Omron CX-Programmer project NewProject (CX-Programmer 9.80)

# PLC NewPLC1: CQM1 CPU41

## Program NewProgram1 (no task)

### Section Section1

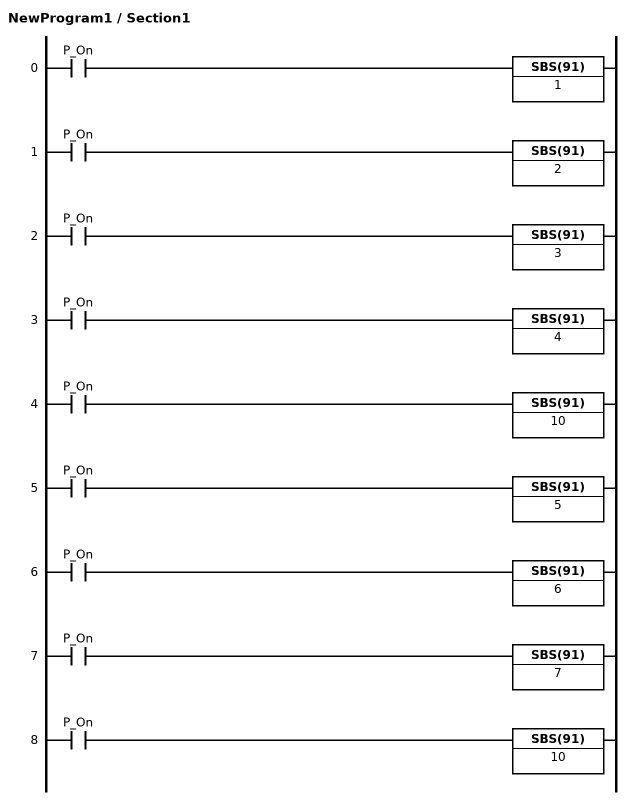
; rung 0
LD P_On
SBS(91) 1
; rung 1
LD P_On
SBS(91) 2
; rung 2
LD P_On
SBS(91) 3
; rung 3
LD P_On
SBS(91) 4
; rung 4
LD P_On
SBS(91) 10
; rung 5
LD P_On
SBS(91) 5
; rung 6
LD P_On
SBS(91) 6
; rung 7
LD P_On
SBS(91) 7
; rung 8
LD P_On
SBS(91) 10

### Section Section2

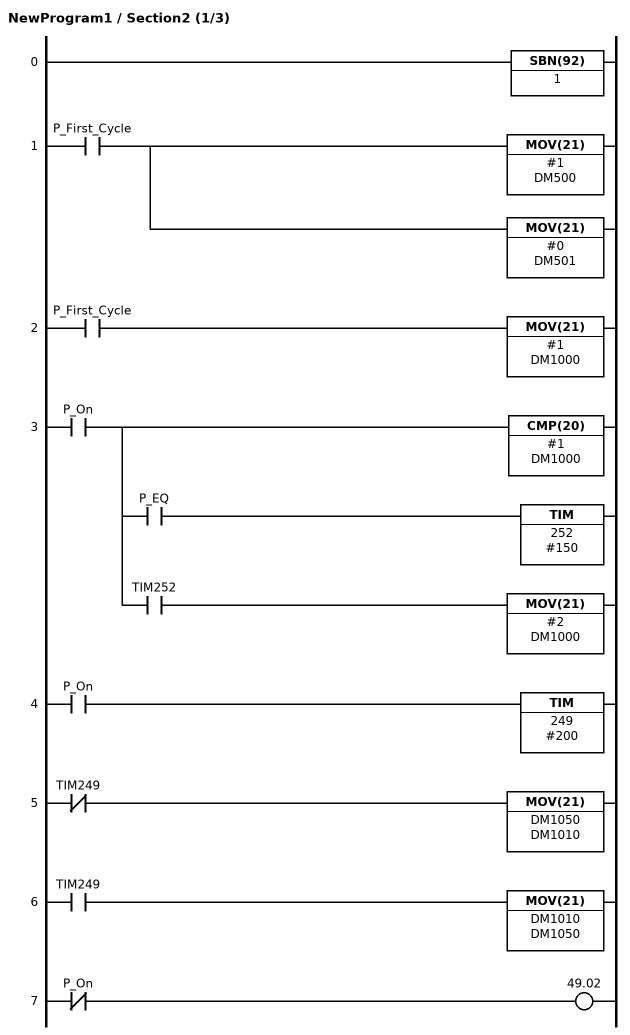
; rung 0
SBN(92) 1
; rung 1
LD P_First_Cycle
MOV(21) #1 DM500
MOV(21) #0 DM501
; rung 2
LD P_First_Cycle
MOV(21) #1 DM1000
; rung 3
LD P_On
OUT TR0
CMP(20) #1 DM1000
AND P_EQ
TIM 252 #150
LD TR0
AND TIM252
MOV(21) #2 DM1000
; rung 4
LD P_On
TIM 249 #200
; rung 5
LDNOT TIM249
MOV(21) DM1050 DM1010
; rung 6
LD TIM249
MOV(21) DM1010 DM1050
; rung 7
LDNOT P_On
OUT 49.02

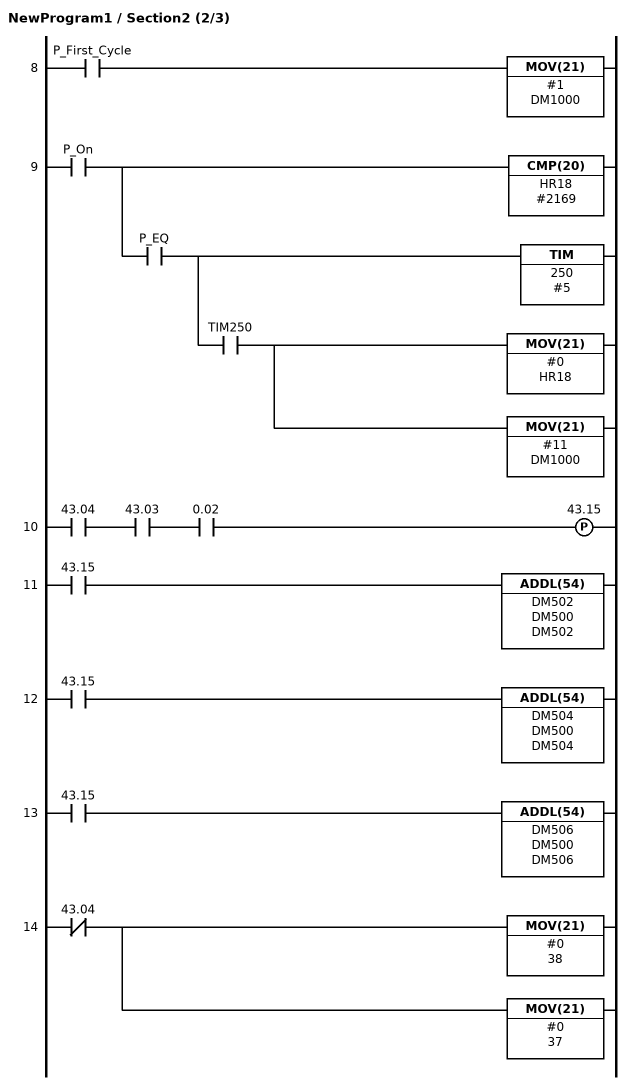
; rung 8
LD P_First_Cycle
MOV(21) #1 DM1000
; rung 9
LD P_On
CMP(20) HR18 #2169
AND P_EQ
TIM 250 #5
AND TIM250
MOV(21) #0 HR18
MOV(21) #11 DM1000
; rung 10
LD 43.04
AND 43.03
AND 0.02
DIFU(13) 43.15
; rung 11
LD 43.15
ADDL(54) DM502 DM500 DM502
; rung 12
LD 43.15
ADDL(54) DM504 DM500 DM504
; rung 13
LD 43.15
ADDL(54) DM506 DM500 DM506
; rung 14
LDNOT 43.04
MOV(21) #0 38
MOV(21) #0 37

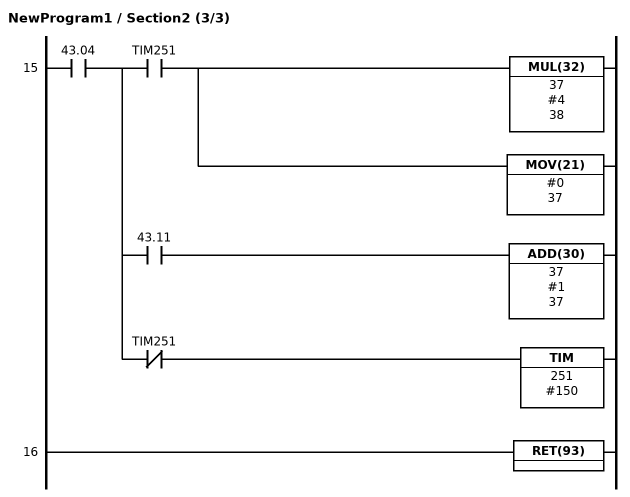
; rung 15
LD 43.04
OUT TR0
AND TIM251
MUL(32) 37 #4 38
MOV(21) #0 37
LD TR0
AND 43.11
ADD(30) 37 #1 37
LD TR0
ANDNOT TIM251
TIM 251 #150
; rung 16
RET(93)

### Section Section3

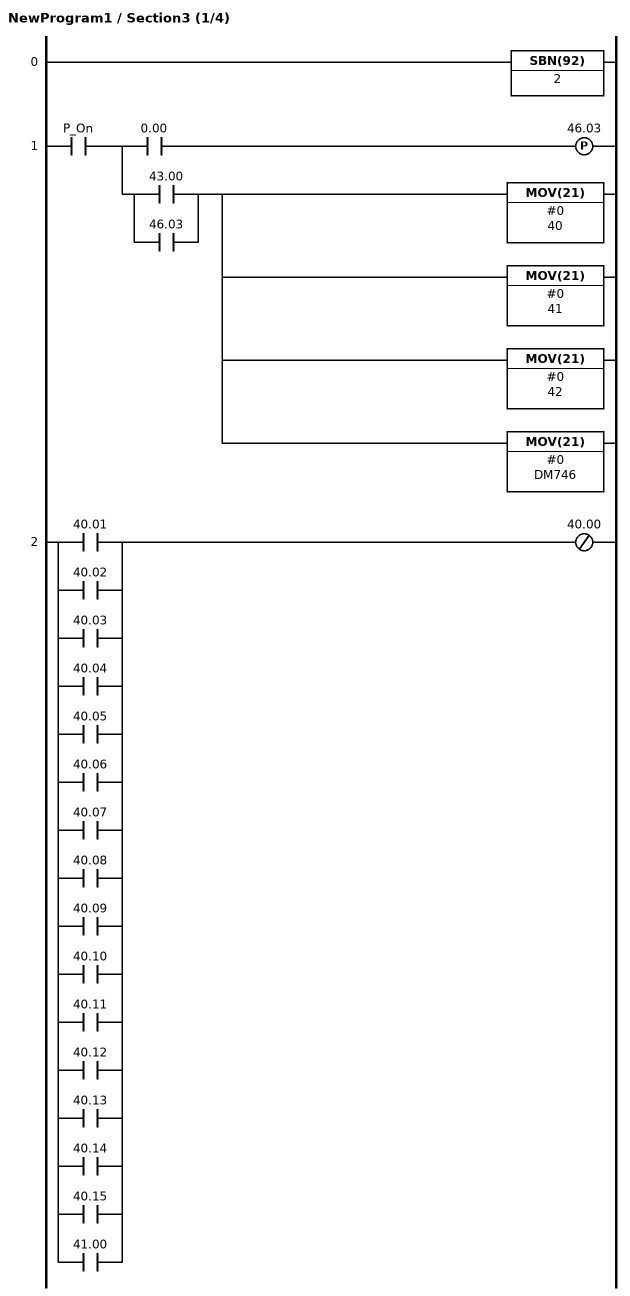
; rung 0
SBN(92) 2
; rung 1
LD P_On
OUT TR0
AND 0.00
DIFU(13) 46.03
LD TR0
LD 43.00
OR 46.03
ANDLD
MOV(21) #0 40
MOV(21) #0 41
MOV(21) #0 42
MOV(21) #0 DM746
; rung 2
LD 40.01
OR 40.02
OR 40.03
OR 40.04
OR 40.05
OR 40.06
OR 40.07
OR 40.08
OR 40.09
OR 40.10
OR 40.11
OR 40.12
OR 40.13
OR 40.14
OR 40.15
OR 41.00
OUTNOT 40.00

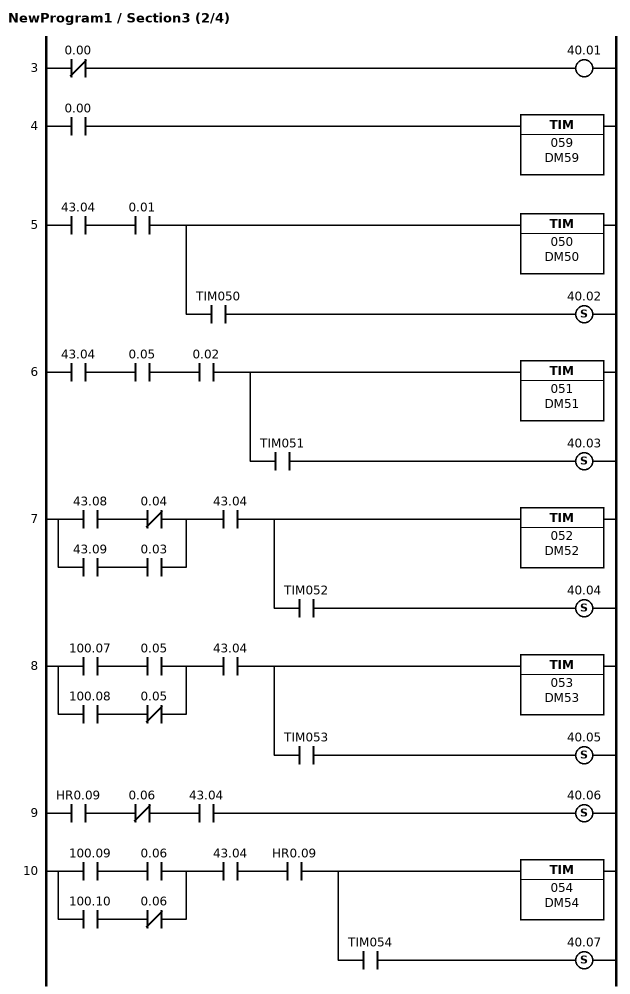
; rung 3
LDNOT 0.00
OUT 40.01
; rung 4
LD 0.00
TIM 059 DM59
; rung 5
LD 43.04
AND 0.01
TIM 050 DM50
AND TIM050
SET 40.02
; rung 6
LD 43.04
AND 0.05
AND 0.02
TIM 051 DM51
AND TIM051
SET 40.03
; rung 7
LD 43.08
ANDNOT 0.04
LD 43.09
AND 0.03
ORLD
AND 43.04
TIM 052 DM52
AND TIM052
SET 40.04
; rung 8
LD 100.07
AND 0.05
LD 100.08
ANDNOT 0.05
ORLD
AND 43.04
TIM 053 DM53
AND TIM053
SET 40.05
; rung 9
LD HR0.09
ANDNOT 0.06
AND 43.04
SET 40.06
; rung 10
LD 100.09
AND 0.06
LD 100.10
ANDNOT 0.06
ORLD
AND 43.04
AND HR0.09
TIM 054 DM54
AND TIM054
SET 40.07

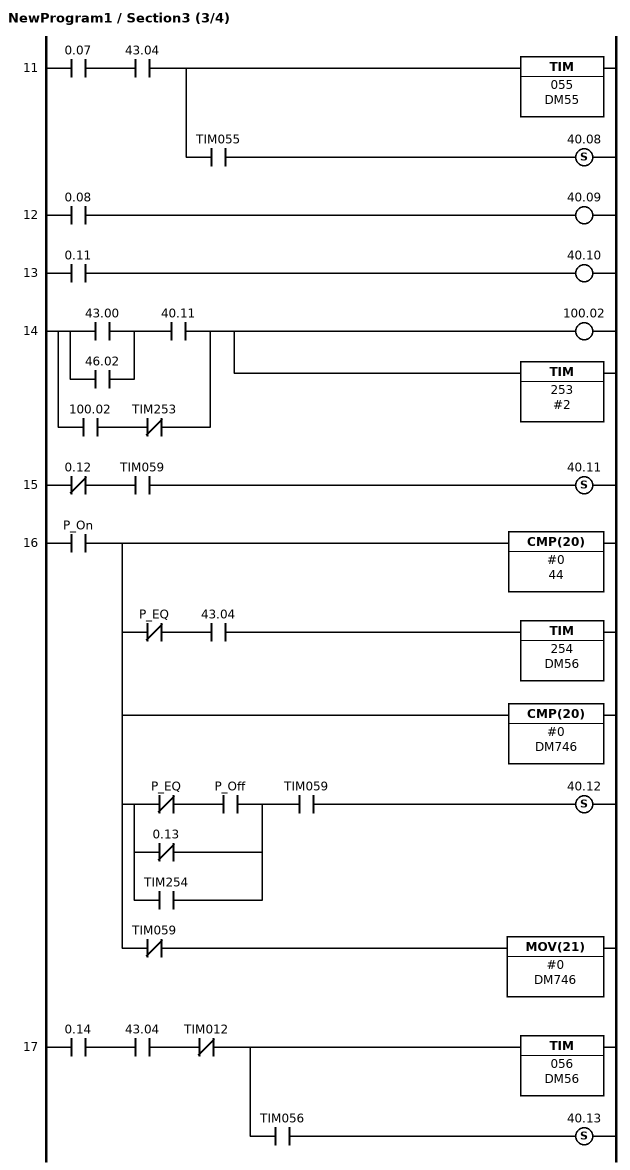
; rung 11
LD 0.07
AND 43.04
TIM 055 DM55
AND TIM055
SET 40.08
; rung 12
LD 0.08
OUT 40.09
; rung 13
LD 0.11
OUT 40.10
; rung 14
LD 43.00
OR 46.02
AND 40.11
LD 100.02
ANDNOT TIM253
ORLD
OUT 100.02
TIM 253 #2
; rung 15
LDNOT 0.12
AND TIM059
SET 40.11
; rung 16
LD P_On
OUT TR0
CMP(20) #0 44
ANDNOT P_EQ
AND 43.04
TIM 254 DM56
LD TR0
CMP(20) #0 DM746
LDNOT P_EQ
AND P_Off
ORNOT 0.13
OR TIM254
ANDLD
AND TIM059
SET 40.12
LD TR0
ANDNOT TIM059
MOV(21) #0 DM746
; rung 17
LD 0.14
AND 43.04
ANDNOT TIM012
TIM 056 DM56
AND TIM056
SET 40.13

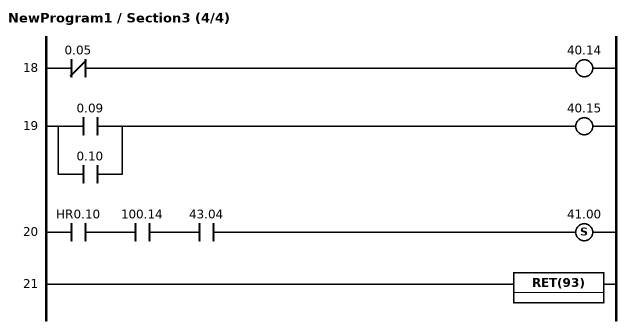
; rung 18
LDNOT 0.05
OUT 40.14
; rung 19
LD 0.09
OR 0.10
OUT 40.15
; rung 20
LD HR0.10
AND 100.14
AND 43.04
SET 41.00
; rung 21
RET(93)

### Section Section4

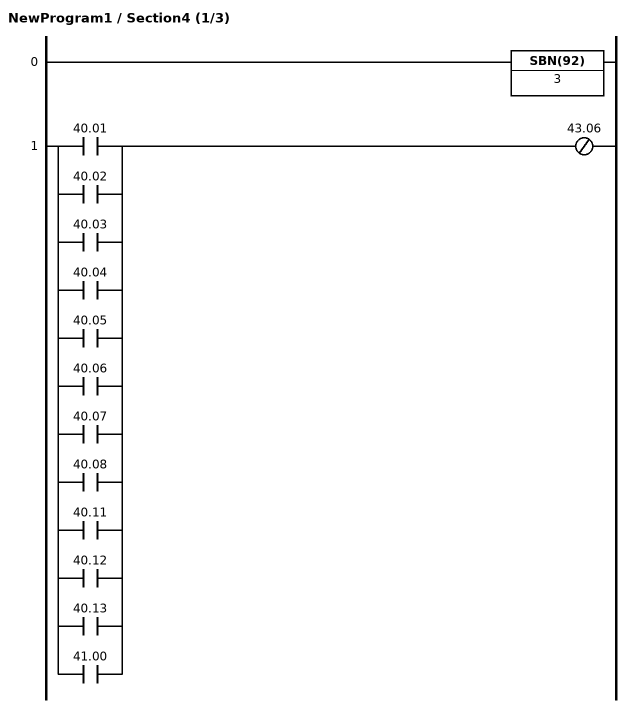
; rung 0
SBN(92) 3
; rung 1
LD 40.01
OR 40.02
OR 40.03
OR 40.04
OR 40.05
OR 40.06
OR 40.07
OR 40.08
OR 40.11
OR 40.12
OR 40.13
OR 41.00
OUTNOT 43.06

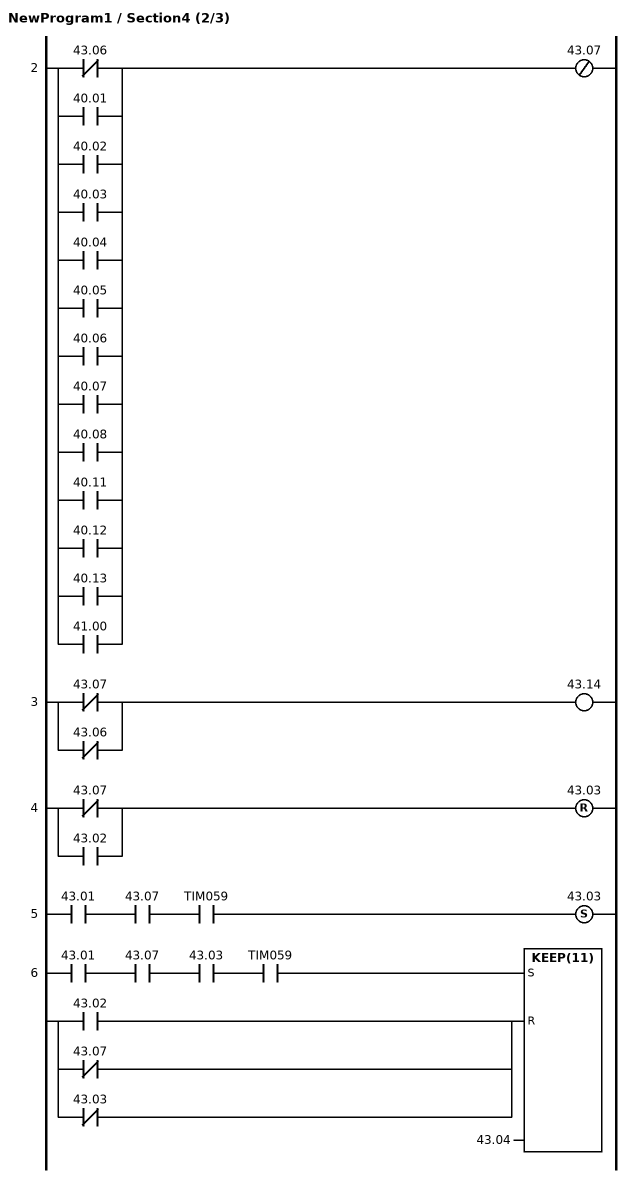
; rung 2
LDNOT 43.06
OR 40.01
OR 40.02
OR 40.03
OR 40.04
OR 40.05
OR 40.06
OR 40.07
OR 40.08
OR 40.11
OR 40.12
OR 40.13
OR 41.00
OUTNOT 43.07
; rung 3
LDNOT 43.07
ORNOT 43.06
OUT 43.14
; rung 4
LDNOT 43.07
OR 43.02
RSET 43.03
; rung 5
LD 43.01
AND 43.07
AND TIM059
SET 43.03
; rung 6
LD 43.01
AND 43.07
AND 43.03
AND TIM059
LD 43.02
ORNOT 43.07
ORNOT 43.03
KEEP(11) 43.04

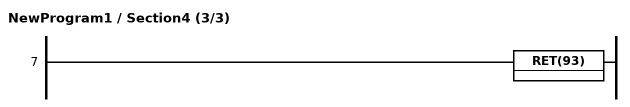
; rung 7
RET(93)

### Section Section5

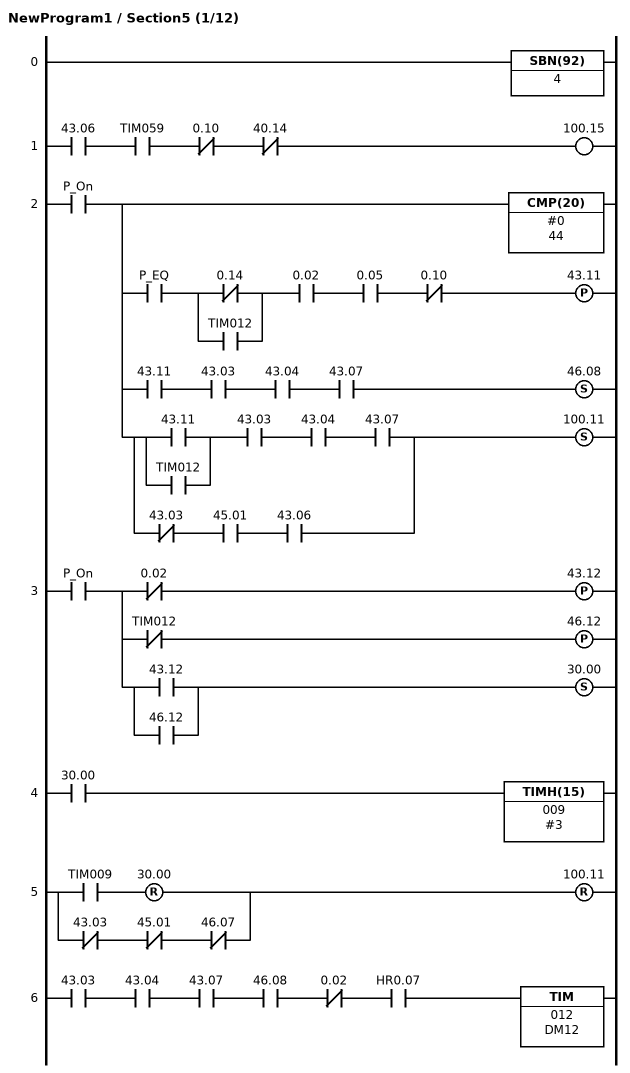
; rung 0
SBN(92) 4
; rung 1
LD 43.06
AND TIM059
ANDNOT 0.10
ANDNOT 40.14
OUT 100.15
; rung 2
LD P_On
OUT TR0
CMP(20) #0 44
AND P_EQ
LDNOT 0.14
OR TIM012
ANDLD
AND 0.02
AND 0.05
ANDNOT 0.10
DIFU(13) 43.11
LD TR0
AND 43.11
AND 43.03
AND 43.04
AND 43.07
SET 46.08
LD TR0
LD 43.11
OR TIM012
AND 43.03
AND 43.04
AND 43.07
LDNOT 43.03
AND 45.01
AND 43.06
ORLD
ANDLD
SET 100.11
; rung 3
LD P_On
OUT TR0
ANDNOT 0.02
DIFU(13) 43.12
LD TR0
ANDNOT TIM012
DIFU(13) 46.12
LD TR0
LD 43.12
OR 46.12
ANDLD
SET 30.00
; rung 4
LD 30.00
TIMH(15) 009 #3
; rung 5
LD TIM009
RSET 30.00
LDNOT 43.03
ANDNOT 45.01
ANDNOT 46.07
ORLD
RSET 100.11
; rung 6
LD 43.03
AND 43.04
AND 43.07
AND 46.08
ANDNOT 0.02
AND HR0.07
TIM 012 DM12

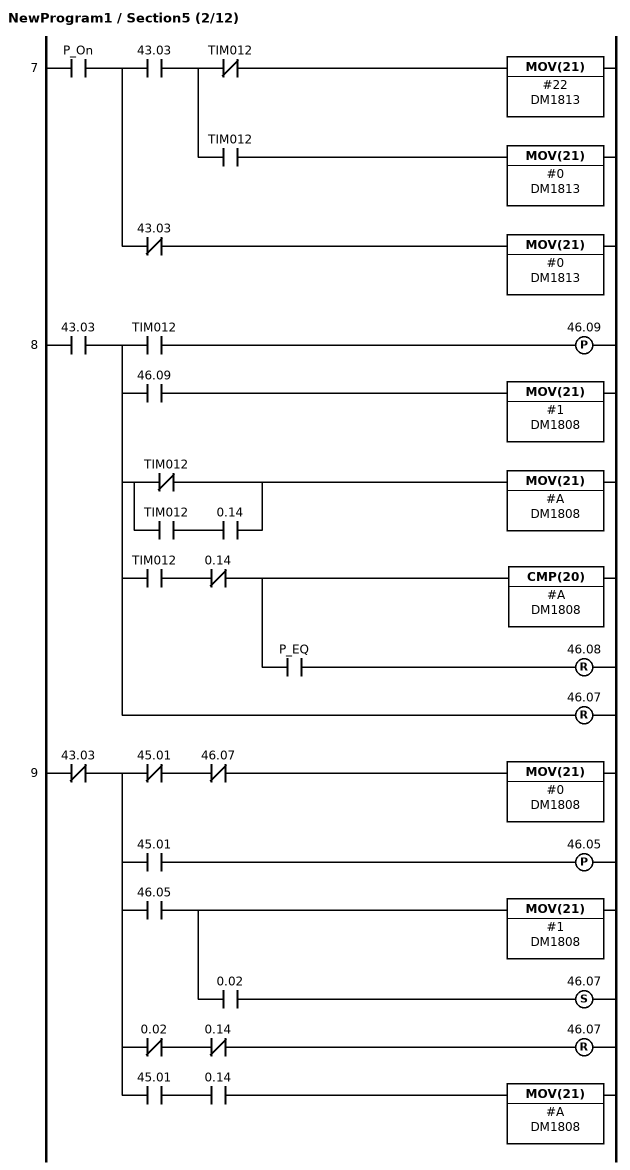
; rung 7
LD P_On
OUT TR0
AND 43.03
OUT TR1
ANDNOT TIM012
MOV(21) #22 DM1813
LD TR1
AND TIM012
MOV(21) #0 DM1813
LD TR0
ANDNOT 43.03
MOV(21) #0 DM1813
; rung 8
LD 43.03
OUT TR0
AND TIM012
DIFU(13) 46.09
LD TR0
AND 46.09
MOV(21) #1 DM1808
LD TR0
LDNOT TIM012
LD TIM012
AND 0.14
ORLD
ANDLD
MOV(21) #A DM1808
LD TR0
AND TIM012
ANDNOT 0.14
CMP(20) #A DM1808
AND P_EQ
RSET 46.08
LD TR0
RSET 46.07
; rung 9
LDNOT 43.03
OUT TR0
ANDNOT 45.01
ANDNOT 46.07
MOV(21) #0 DM1808
LD TR0
AND 45.01
DIFU(13) 46.05
LD TR0
AND 46.05
MOV(21) #1 DM1808
AND 0.02
SET 46.07
LD TR0
ANDNOT 0.02
ANDNOT 0.14
RSET 46.07
LD TR0
AND 45.01
AND 0.14
MOV(21) #A DM1808

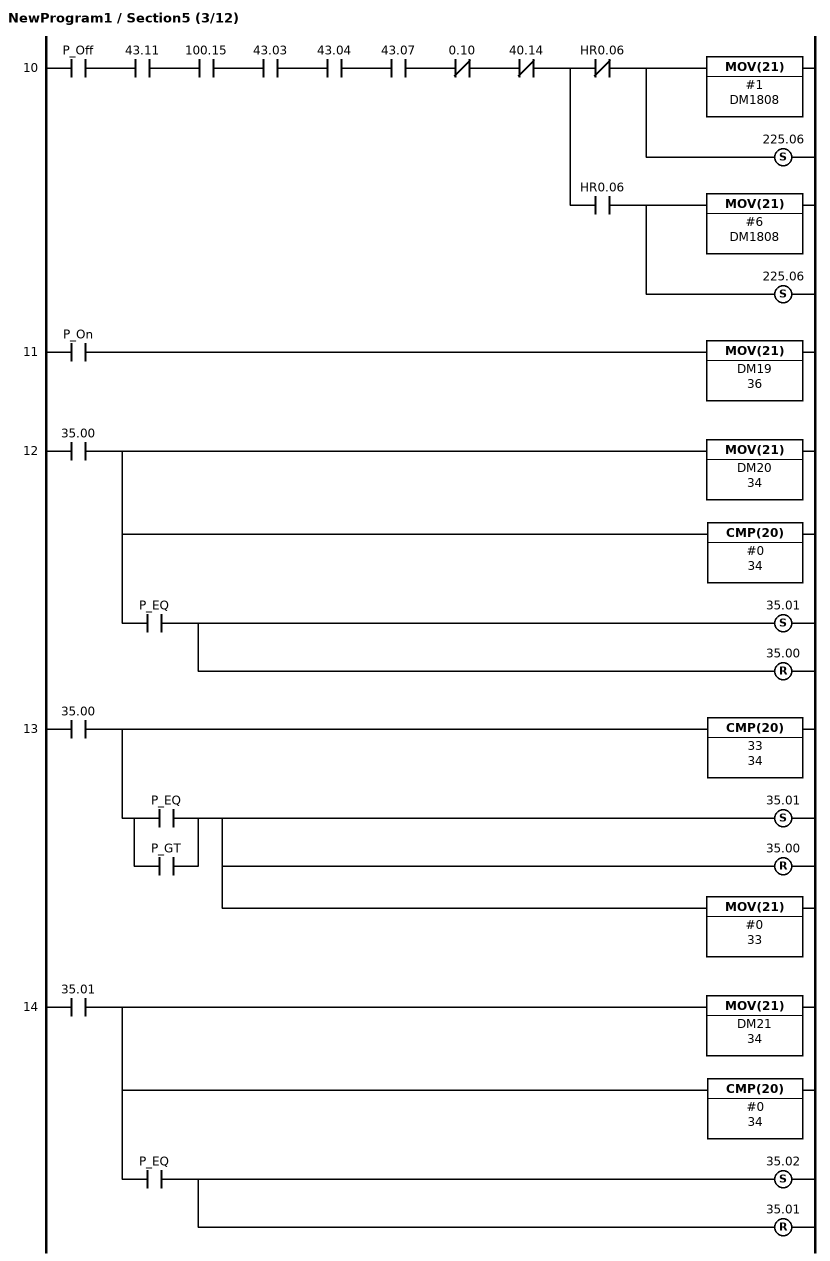
; rung 10
LD P_Off
AND 43.11
AND 100.15
AND 43.03
AND 43.04
AND 43.07
ANDNOT 0.10
ANDNOT 40.14
OUT TR0
ANDNOT HR0.06
MOV(21) #1 DM1808
SET 225.06
LD TR0
AND HR0.06
MOV(21) #6 DM1808
SET 225.06
; rung 11
LD P_On
MOV(21) DM19 36
; rung 12
LD 35.00
MOV(21) DM20 34
CMP(20) #0 34
AND P_EQ
SET 35.01
RSET 35.00
; rung 13
LD 35.00
CMP(20) 33 34
LD P_EQ
OR P_GT
ANDLD
SET 35.01
RSET 35.00
MOV(21) #0 33
; rung 14
LD 35.01
MOV(21) DM21 34
CMP(20) #0 34
AND P_EQ
SET 35.02
RSET 35.01

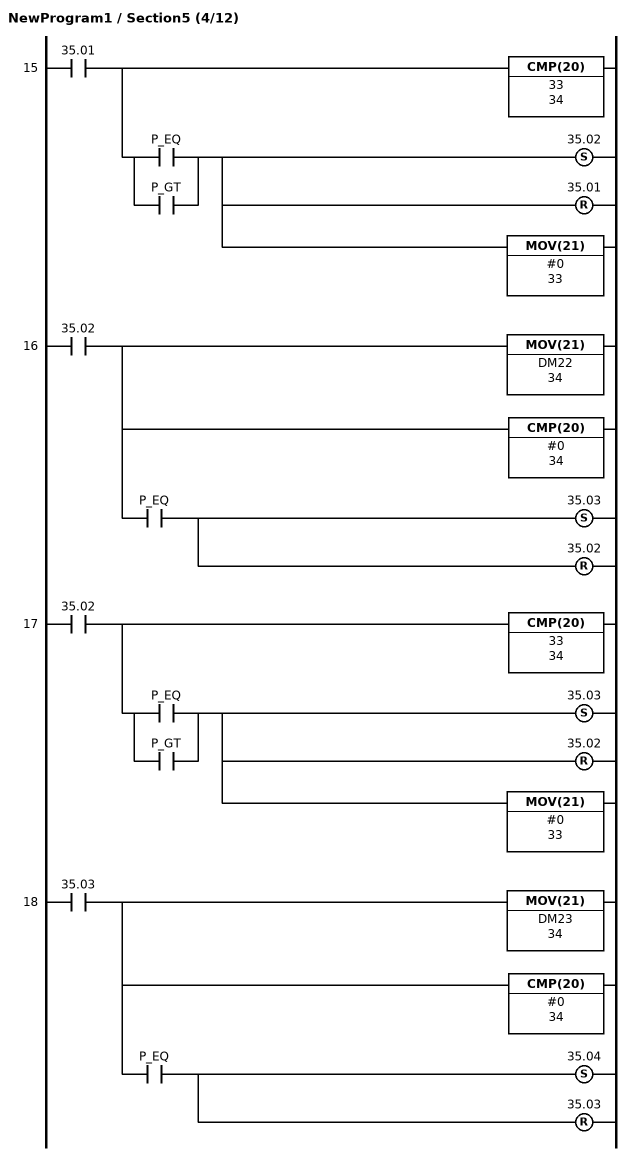
; rung 15
LD 35.01
CMP(20) 33 34
LD P_EQ
OR P_GT
ANDLD
SET 35.02
RSET 35.01
MOV(21) #0 33
; rung 16
LD 35.02
MOV(21) DM22 34
CMP(20) #0 34
AND P_EQ
SET 35.03
RSET 35.02
; rung 17
LD 35.02
CMP(20) 33 34
LD P_EQ
OR P_GT
ANDLD
SET 35.03
RSET 35.02
MOV(21) #0 33
; rung 18
LD 35.03
MOV(21) DM23 34
CMP(20) #0 34
AND P_EQ
SET 35.04
RSET 35.03

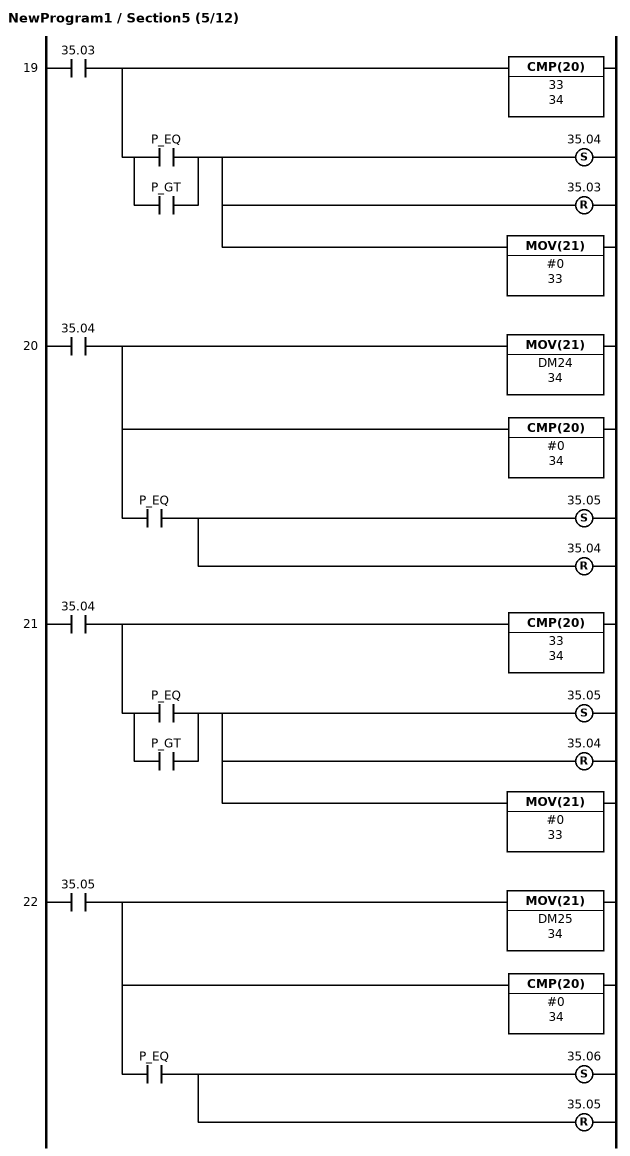
; rung 19
LD 35.03
CMP(20) 33 34
LD P_EQ
OR P_GT
ANDLD
SET 35.04
RSET 35.03
MOV(21) #0 33
; rung 20
LD 35.04
MOV(21) DM24 34
CMP(20) #0 34
AND P_EQ
SET 35.05
RSET 35.04
; rung 21
LD 35.04
CMP(20) 33 34
LD P_EQ
OR P_GT
ANDLD
SET 35.05
RSET 35.04
MOV(21) #0 33
; rung 22
LD 35.05
MOV(21) DM25 34
CMP(20) #0 34
AND P_EQ
SET 35.06
RSET 35.05

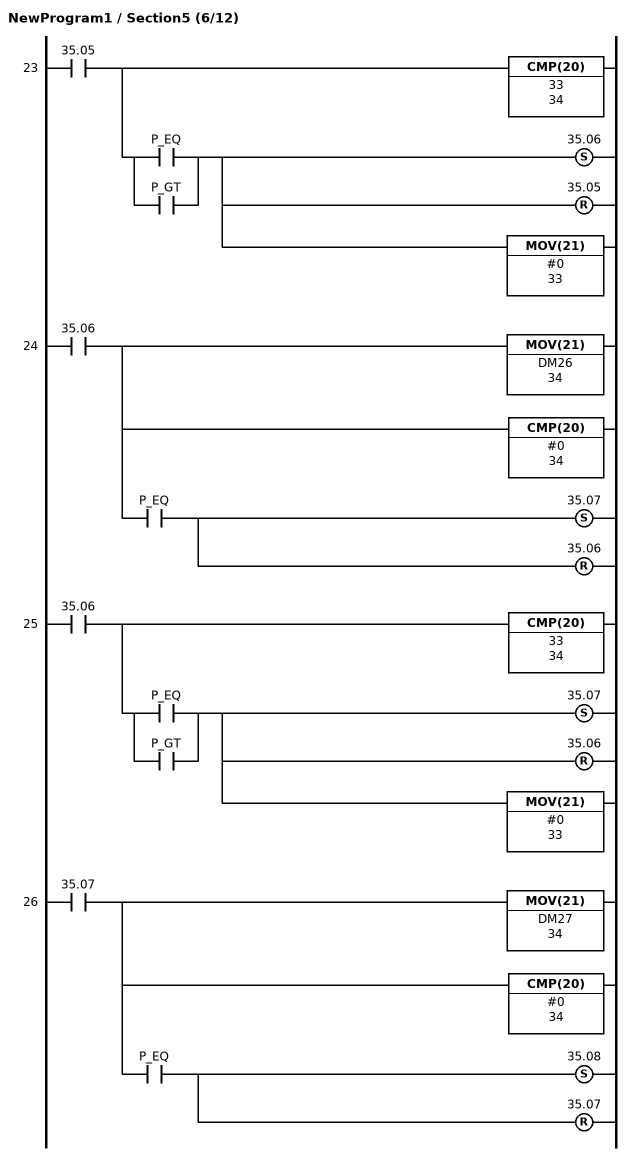
; rung 23
LD 35.05
CMP(20) 33 34
LD P_EQ
OR P_GT
ANDLD
SET 35.06
RSET 35.05
MOV(21) #0 33
; rung 24
LD 35.06
MOV(21) DM26 34
CMP(20) #0 34
AND P_EQ
SET 35.07
RSET 35.06
; rung 25
LD 35.06
CMP(20) 33 34
LD P_EQ
OR P_GT
ANDLD
SET 35.07
RSET 35.06
MOV(21) #0 33
; rung 26
LD 35.07
MOV(21) DM27 34
CMP(20) #0 34
AND P_EQ
SET 35.08
RSET 35.07

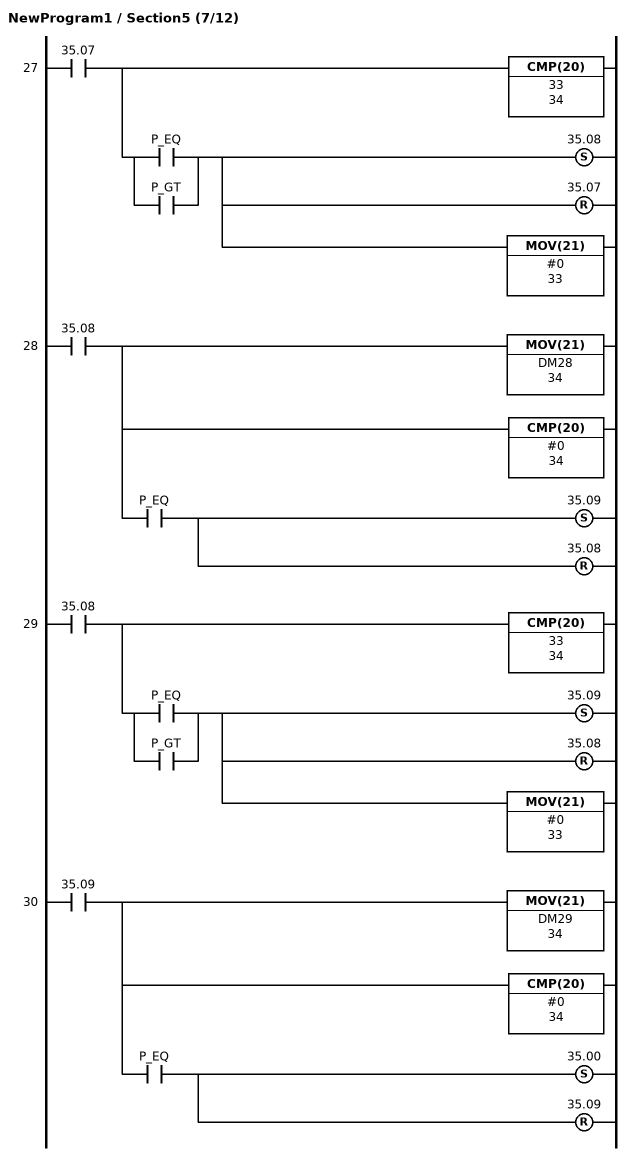
; rung 27
LD 35.07
CMP(20) 33 34
LD P_EQ
OR P_GT
ANDLD
SET 35.08
RSET 35.07
MOV(21) #0 33
; rung 28
LD 35.08
MOV(21) DM28 34
CMP(20) #0 34
AND P_EQ
SET 35.09
RSET 35.08
; rung 29
LD 35.08
CMP(20) 33 34
LD P_EQ
OR P_GT
ANDLD
SET 35.09
RSET 35.08
MOV(21) #0 33
; rung 30
LD 35.09
MOV(21) DM29 34
CMP(20) #0 34
AND P_EQ
SET 35.00
RSET 35.09

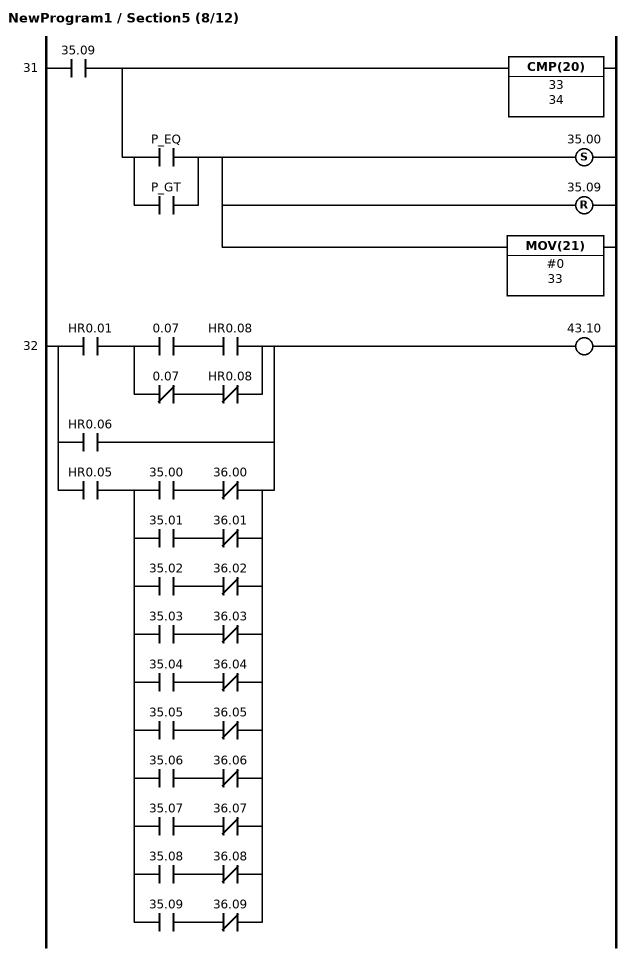
; rung 31
LD 35.09
CMP(20) 33 34
LD P_EQ
OR P_GT
ANDLD
SET 35.00
RSET 35.09
MOV(21) #0 33
; rung 32
LD HR0.01
LD 0.07
AND HR0.08
LDNOT 0.07
ANDNOT HR0.08
ORLD
ANDLD
OR HR0.06
LD HR0.05
LD 35.00
ANDNOT 36.00
LD 35.01
ANDNOT 36.01
ORLD
LD 35.02
ANDNOT 36.02
ORLD
LD 35.03
ANDNOT 36.03
ORLD
LD 35.04
ANDNOT 36.04
ORLD
LD 35.05
ANDNOT 36.05
ORLD
LD 35.06
ANDNOT 36.06
ORLD
LD 35.07
ANDNOT 36.07
ORLD
LD 35.08
ANDNOT 36.08
ORLD
LD 35.09
ANDNOT 36.09
ORLD
ANDLD
ORLD
OUT 43.10

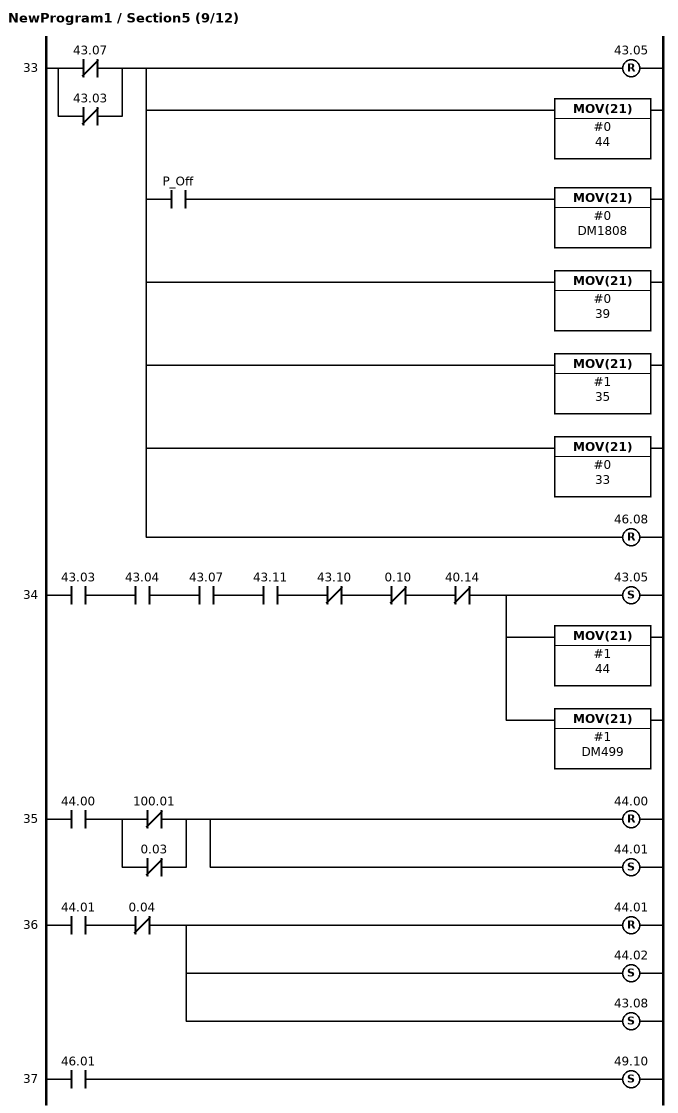
; rung 33
LDNOT 43.07
ORNOT 43.03
OUT TR0
RSET 43.05
MOV(21) #0 44
AND P_Off
MOV(21) #0 DM1808
LD TR0
MOV(21) #0 39
MOV(21) #1 35
MOV(21) #0 33
RSET 46.08
; rung 34
LD 43.03
AND 43.04
AND 43.07
AND 43.11
ANDNOT 43.10
ANDNOT 0.10
ANDNOT 40.14
SET 43.05
MOV(21) #1 44
MOV(21) #1 DM499
; rung 35
LD 44.00
LDNOT 100.01
ORNOT 0.03
ANDLD
RSET 44.00
SET 44.01
; rung 36
LD 44.01
ANDNOT 0.04
RSET 44.01
SET 44.02
SET 43.08
; rung 37
LD 46.01
SET 49.10

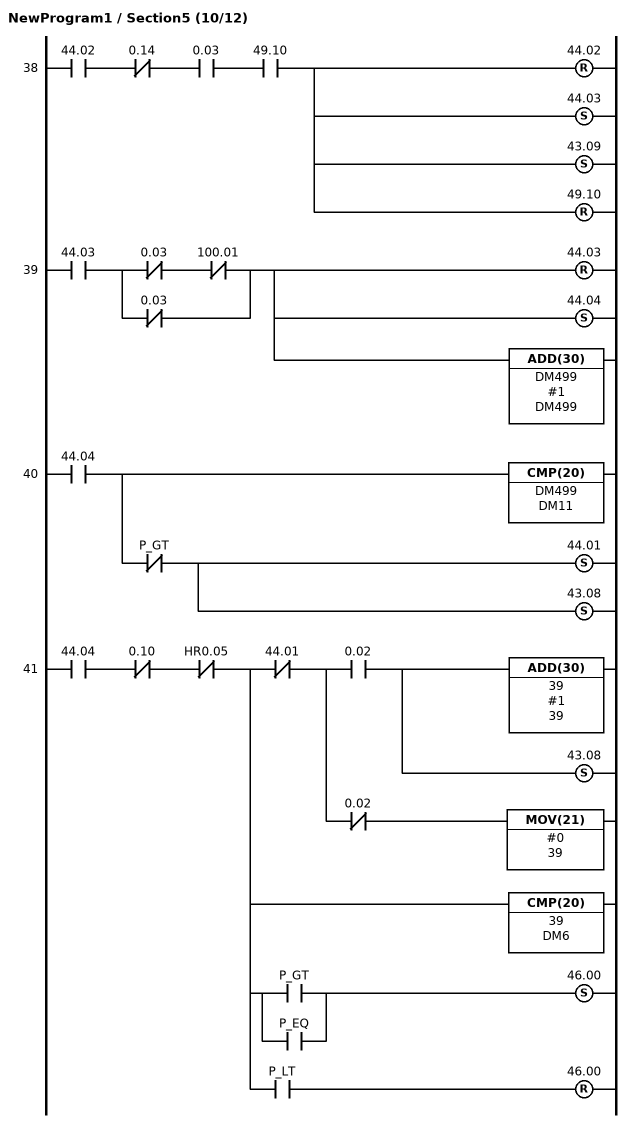
; rung 38
LD 44.02
ANDNOT 0.14
AND 0.03
AND 49.10
RSET 44.02
SET 44.03
SET 43.09
RSET 49.10
; rung 39
LD 44.03
LDNOT 0.03
ANDNOT 100.01
ORNOT 0.03
ANDLD
RSET 44.03
SET 44.04
ADD(30) DM499 #1 DM499
; rung 40
LD 44.04
CMP(20) DM499 DM11
ANDNOT P_GT
SET 44.01
SET 43.08
; rung 41
LD 44.04
ANDNOT 0.10
ANDNOT HR0.05
OUT TR0
ANDNOT 44.01
OUT TR1
AND 0.02
ADD(30) 39 #1 39
SET 43.08
LD TR1
ANDNOT 0.02
MOV(21) #0 39
LD TR0
CMP(20) 39 DM6
LD P_GT
OR P_EQ
ANDLD
SET 46.00
LD TR0
AND P_LT
RSET 46.00

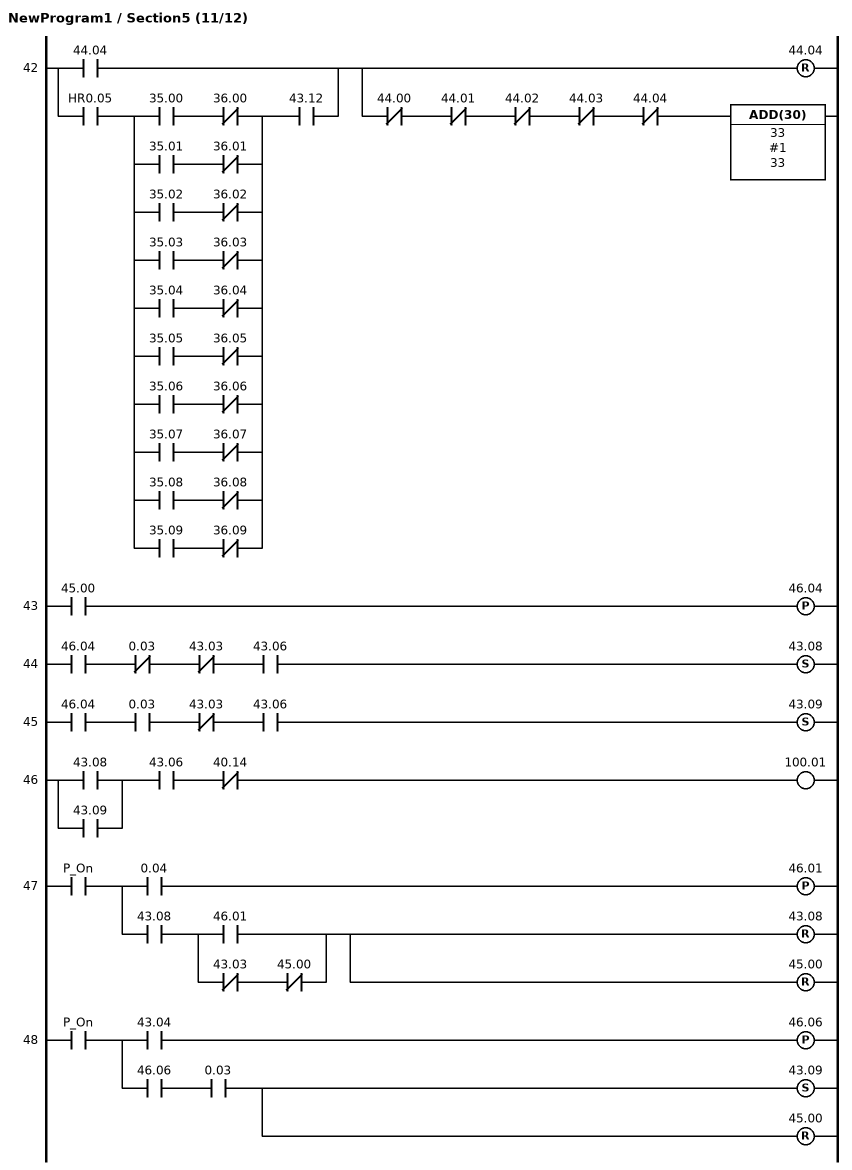
; rung 42
LD 44.04
LD HR0.05
LD 35.00
ANDNOT 36.00
LD 35.01
ANDNOT 36.01
ORLD
LD 35.02
ANDNOT 36.02
ORLD
LD 35.03
ANDNOT 36.03
ORLD
LD 35.04
ANDNOT 36.04
ORLD
LD 35.05
ANDNOT 36.05
ORLD
LD 35.06
ANDNOT 36.06
ORLD
LD 35.07
ANDNOT 36.07
ORLD
LD 35.08
ANDNOT 36.08
ORLD
LD 35.09
ANDNOT 36.09
ORLD
ANDLD
AND 43.12
ORLD
RSET 44.04
ANDNOT 44.00
ANDNOT 44.01
ANDNOT 44.02
ANDNOT 44.03
ANDNOT 44.04
ADD(30) 33 #1 33
; rung 43
LD 45.00
DIFU(13) 46.04
; rung 44
LD 46.04
ANDNOT 0.03
ANDNOT 43.03
AND 43.06
SET 43.08
; rung 45
LD 46.04
AND 0.03
ANDNOT 43.03
AND 43.06
SET 43.09
; rung 46
LD 43.08
OR 43.09
AND 43.06
ANDNOT 40.14
OUT 100.01
; rung 47
LD P_On
OUT TR0
AND 0.04
DIFU(13) 46.01
LD TR0
AND 43.08
LD 46.01
LDNOT 43.03
ANDNOT 45.00
ORLD
ANDLD
RSET 43.08
RSET 45.00
; rung 48
LD P_On
OUT TR0
AND 43.04
DIFU(13) 46.06
LD TR0
AND 46.06
AND 0.03
SET 43.09
RSET 45.00

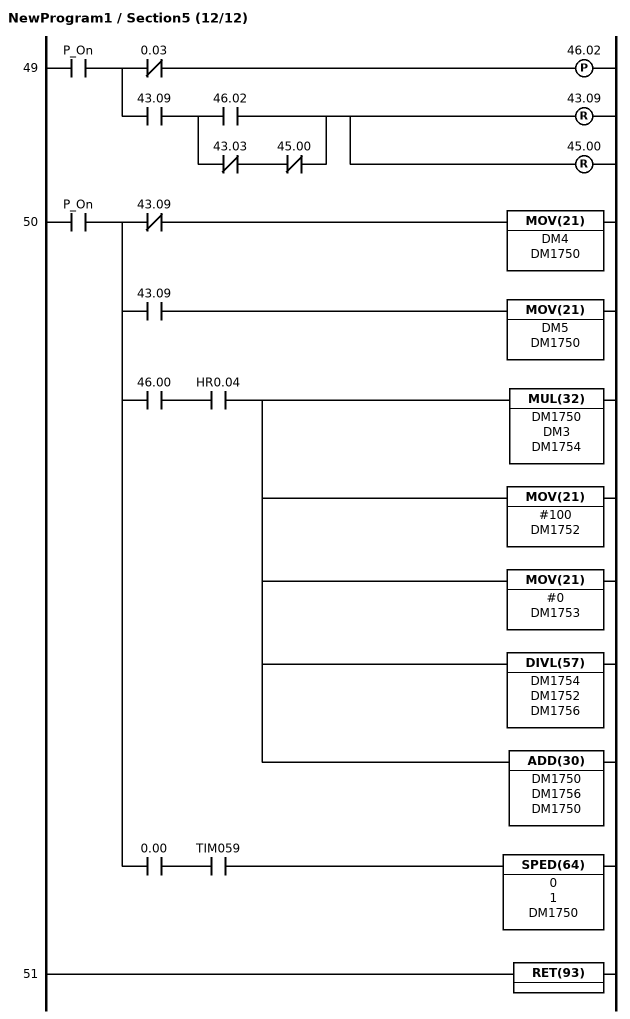
; rung 49
LD P_On
OUT TR0
ANDNOT 0.03
DIFU(13) 46.02
LD TR0
AND 43.09
LD 46.02
LDNOT 43.03
ANDNOT 45.00
ORLD
ANDLD
RSET 43.09
RSET 45.00
; rung 50
LD P_On
OUT TR0
ANDNOT 43.09
MOV(21) DM4 DM1750
LD TR0
AND 43.09
MOV(21) DM5 DM1750
LD TR0
AND 46.00
AND HR0.04
MUL(32) DM1750 DM3 DM1754
MOV(21) #100 DM1752
MOV(21) #0 DM1753
DIVL(57) DM1754 DM1752 DM1756
ADD(30) DM1750 DM1756 DM1750
LD TR0
AND 0.00
AND TIM059
SPED(64) 0 1 DM1750
; rung 51
RET(93)

### Section Section6

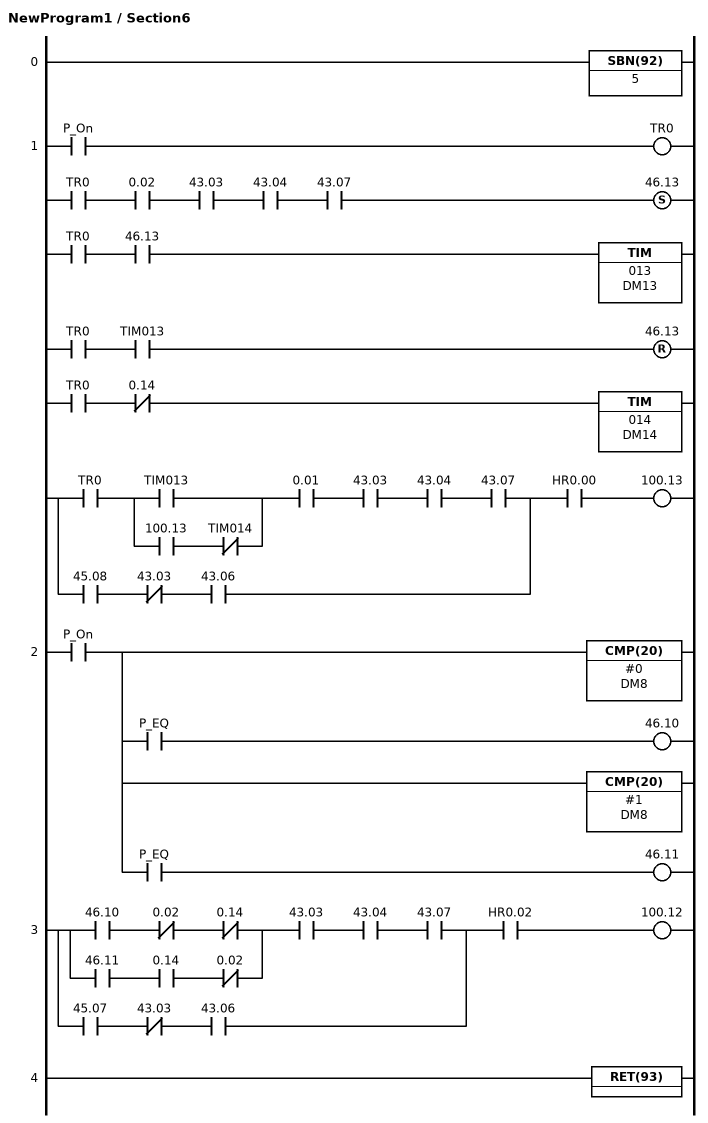
; rung 0
SBN(92) 5
; rung 1
LD P_On
OUT TR0
AND 0.02
AND 43.03
AND 43.04
AND 43.07
SET 46.13
LD TR0
AND 46.13
TIM 013 DM13
LD TR0
AND TIM013
RSET 46.13
LD TR0
ANDNOT 0.14
TIM 014 DM14
LD TR0
LD TIM013
LD 100.13
ANDNOT TIM014
ORLD
ANDLD
AND 0.01
AND 43.03
AND 43.04
AND 43.07
LD 45.08
ANDNOT 43.03
AND 43.06
ORLD
AND HR0.00
OUT 100.13
; rung 2
LD P_On
OUT TR0
CMP(20) #0 DM8
AND P_EQ
OUT 46.10
LD TR0
CMP(20) #1 DM8
AND P_EQ
OUT 46.11
; rung 3
LD 46.10
ANDNOT 0.02
ANDNOT 0.14
LD 46.11
AND 0.14
ANDNOT 0.02
ORLD
AND 43.03
AND 43.04
AND 43.07
LD 45.07
ANDNOT 43.03
AND 43.06
ORLD
AND HR0.02
OUT 100.12
; rung 4
RET(93)

### Section Section7

